TEXTLIST BCF_Version
  Version = 'R1.12.0'
  Company = 'Swisslog'
   = ''
END_TEXTLIST

(* stored: Version 1.1.0.1, ProductVersion 3.1.4024.4
   TextList BCF_Version: Id {391185ce-39f7-4c13-ba86-22460e8183ea} *)
